// TIA Portal V18 export
// export: Created 2026-01-09T11:31:59.6911216Z, ExportSetting WithDefaults, DisplayName Totally Integrated Automation Portal, DisplayVersion V18 Update 5, DisplayName TIA Portal Openness, DisplayVersion V18 Update 5, DisplayName TIA Portal Teamcenter Gateway, DisplayVersion V18, DisplayName TIA Portal Version Control Interface, DisplayVersion V18, DisplayName SINAMICS Startdrive Advanced, DisplayVersion V18 SP2 Update 1, DisplayName SINAMICS Startdrive G110M, G120, G120C, G120D, G120P, G115D, DisplayVersion V18 SP2 Update 1, DisplayName SINAMICS Startdrive G130, G150, S120, S150, SINAMICS MV, S210, G220, S200, DisplayVersion V18 SP2 Update 1, DisplayName STEP 7 Professional, DisplayVersion V18 Update 5, DisplayName STEP 7 Safety, DisplayVersion V18, DisplayName WinCC Professional, DisplayVersion V18 Update 5
TagTable "2Command Mes To PLC_DB501"
  MEStoPLC_Load_Station1PartOK : Bool  (PLC tag MEStoPLC."MES.Load_Station1PartOK", CPU S71500-2PN_TP700, 1 s)
  MEStoPLC_Load_Station1PartNG : Bool  (PLC tag MEStoPLC."MES.Load_Station1PartNG", CPU S71500-2PN_TP700, 1 s)
  MEStoPLC_Load_Station1ReqMesDone : Bool  (PLC tag MEStoPLC."MES.Load_Station1ReqMesDone", CPU S71500-2PN_TP700, 1 s)
  MEStoPLC_Load_Station1Spare : Bool  (PLC tag MEStoPLC.Spare_1, CPU S71500-2PN_TP700, 1 s)
  MEStoPLC_Load_Station1Spare1 : Bool  (PLC tag MEStoPLC."MES.Load_Station2PartOK", CPU S71500-2PN_TP700, 1 s)
  MEStoPLC_Load_Station1Spare2 : Bool  (PLC tag MEStoPLC."MES.Load_Station2PartNG", CPU S71500-2PN_TP700, 1 s)
  MEStoPLC_Load_Station1Spare3 : Bool  (PLC tag MEStoPLC."MES.Load_Station2ReqMesDone", CPU S71500-2PN_TP700, 1 s)
  MEStoPLC_Load_Station1Spare4 : Bool  (PLC tag MEStoPLC.Spare_2, CPU S71500-2PN_TP700, 1 s)
  MEStoPLC_Load_Station2PartOK : Bool  (PLC tag MEStoPLC."MES.Load_Station3PartOK", CPU S71500-2PN_TP700, 1 s)
  MEStoPLC_Load_Station2PartNG : Bool  (PLC tag MEStoPLC."MES.Load_Station3PartNG", CPU S71500-2PN_TP700, 1 s)
  MEStoPLC_Load_Station2ReqMesDone : Bool  (PLC tag MEStoPLC."MES.Load_Station3ReqMesDone", CPU S71500-2PN_TP700, 1 s)
  MEStoPLC_Load_Station2Spare : Bool  (PLC tag MEStoPLC.Spare_3, CPU S71500-2PN_TP700, 1 s)
  MEStoPLC_Load_Station2Spare1 : Bool  (PLC tag MEStoPLC."MES.Load_Station4PartOK", CPU S71500-2PN_TP700, 1 s)
  MEStoPLC_Load_Station2Spare2 : Bool  (PLC tag MEStoPLC."MES.Load_Station4PartNG", CPU S71500-2PN_TP700, 1 s)
  MEStoPLC_Load_Station2Spare3 : Bool  (PLC tag MEStoPLC."MES.Load_Station4ReqMesDone", CPU S71500-2PN_TP700, 1 s)
  MEStoPLC_Load_Station2Spare4 : Bool  (PLC tag MEStoPLC.Spare_4, CPU S71500-2PN_TP700, 1 s)
  MEStoPLC_Load_Station3PartOK : Bool  (PLC tag MEStoPLC."MES.Load_Station5PartOK", CPU S71500-2PN_TP700, 1 s)
  MEStoPLC_Load_Station3PartNG : Bool  (PLC tag MEStoPLC."MES.Load_Station5PartNG", CPU S71500-2PN_TP700, 1 s)
  MEStoPLC_Load_Station3ReqMesDone : Bool  (PLC tag MEStoPLC."MES.Load_Station5ReqMesDone", CPU S71500-2PN_TP700, 1 s)
  MEStoPLC_Load_Station3Spare : Bool  (PLC tag MEStoPLC.Spare_5, CPU S71500-2PN_TP700, 1 s)
  MEStoPLC_Load_Station3Spare1 : Bool  (PLC tag MEStoPLC."MES.Load_Station6PartOK", CPU S71500-2PN_TP700, 1 s)
  MEStoPLC_Load_Station3Spare2 : Bool  (PLC tag MEStoPLC."MES.Load_Station6PartNG", CPU S71500-2PN_TP700, 1 s)
  MEStoPLC_Load_Station3Spare3 : Bool  (PLC tag MEStoPLC."MES.Load_Station6ReqMesDone", CPU S71500-2PN_TP700, 1 s)
  MEStoPLC_Load_Station3Spare4 : Bool  (PLC tag MEStoPLC.Spare_6, CPU S71500-2PN_TP700, 1 s)
  MEStoPLC_Load_Station4PartOK : Bool  (PLC tag MEStoPLC."MES.Load_Station7PartOK", CPU S71500-2PN_TP700, 1 s)
  MEStoPLC_Load_Station4PartNG : Bool  (PLC tag MEStoPLC."MES.Load_Station7PartNG", CPU S71500-2PN_TP700, 1 s)
  MEStoPLC_Load_Station4ReqMesDone : Bool  (PLC tag MEStoPLC."MES.Load_Station7ReqMesDone", CPU S71500-2PN_TP700, 1 s)
  MEStoPLC_Load_Station4Spare : Bool  (PLC tag MEStoPLC.Spare_7, CPU S71500-2PN_TP700, 1 s)
  MEStoPLC_Load_Station4Spare1 : Bool  (PLC tag MEStoPLC."MES.Load_Station8PartOK", CPU S71500-2PN_TP700, 1 s)
  MEStoPLC_Load_Station4Spare2 : Bool  (PLC tag MEStoPLC."MES.Load_Station8PartNG", CPU S71500-2PN_TP700, 1 s)
  MEStoPLC_Load_Station4Spare3 : Bool  (PLC tag MEStoPLC."MES.Load_Station8ReqMesDone", CPU S71500-2PN_TP700, 1 s)
  MEStoPLC_Load_Station4Spare4 : Bool  (PLC tag MEStoPLC.Spare_8, CPU S71500-2PN_TP700, 1 s)
  MEStoPLC_Load_Station5PartOK : Bool  (PLC tag MEStoPLC.Spare_9, CPU S71500-2PN_TP700, 1 s)
  MEStoPLC_Load_Station5PartNG : Bool  (PLC tag MEStoPLC.Static_3, CPU S71500-2PN_TP700, 1 s)
  MEStoPLC_Load_Station5ReqMesDone : Bool  (PLC tag MEStoPLC."MES.Load_SubPart1OK", CPU S71500-2PN_TP700, 1 s)
  MEStoPLC_Load_Station5Spare : Bool  (PLC tag MEStoPLC."MES.Load_SubPart1tNG", CPU S71500-2PN_TP700, 1 s)
  MEStoPLC_Load_Station5Spare1 : Bool  (PLC tag MEStoPLC."MES.Load_SubPart1ReqMesDone", CPU S71500-2PN_TP700, 1 s)
  MEStoPLC_Load_Station5Spare2 : Bool  (PLC tag MEStoPLC.Spare_10, CPU S71500-2PN_TP700, 1 s)
  MEStoPLC_Load_Station5Spare3 : Bool  (PLC tag MEStoPLC."MES.Load_SubPart2OK", CPU S71500-2PN_TP700, 1 s)
  MEStoPLC_Load_Station5Spare4 : Bool  (PLC tag MEStoPLC."MES.Load_SubPart2tNG", CPU S71500-2PN_TP700, 1 s)
  MEStoPLC_Load_Station6PartOK : Bool  (PLC tag MEStoPLC."MES.Load_SubPart2ReqMesDone", CPU S71500-2PN_TP700, 1 s)
  MEStoPLC_Load_Station6PartNG : Bool  (PLC tag MEStoPLC.Spare_11, CPU S71500-2PN_TP700, 1 s)
  MEStoPLC_Load_Station6ReqMesDone : Bool  (PLC tag MEStoPLC."MES.Load_SubPart3OK", CPU S71500-2PN_TP700, 1 s)
  MEStoPLC_Load_Station6Spare : Bool  (PLC tag MEStoPLC."MES.Load_SubPart3tNG", CPU S71500-2PN_TP700, 1 s)
  MEStoPLC_Load_Station6Spare1 : Bool  (PLC tag MEStoPLC."MES.Load_SubPart3ReqMesDone", CPU S71500-2PN_TP700, 1 s)
  MEStoPLC_Load_Station6Spare2 : Bool  (PLC tag MEStoPLC.Spare_12, CPU S71500-2PN_TP700, 1 s)
  MEStoPLC_Load_Station6Spare3 : Bool  (PLC tag MEStoPLC."MES.Load_SubPart4OK", CPU S71500-2PN_TP700, 1 s)
  MEStoPLC_Load_Station6Spare4 : Bool  (PLC tag MEStoPLC."MES.Load_SubPart4tNG", CPU S71500-2PN_TP700, 1 s)
  MEStoPLC_Load_Station7PartOK : Bool  (PLC tag MEStoPLC."MES.Load_SubPart4ReqMesDone", CPU S71500-2PN_TP700, 1 s)
  MEStoPLC_Load_Station7PartNG : Bool  (PLC tag MEStoPLC.Spare_13, CPU S71500-2PN_TP700, 1 s)
  MEStoPLC_Load_Station7ReqMesDone : Bool  (PLC tag MEStoPLC."MES.Load_SubPart5OK", CPU S71500-2PN_TP700, 1 s)
  MEStoPLC_Load_Station7Spare : Bool  (PLC tag MEStoPLC."MES.Load_SubPart5tNG", CPU S71500-2PN_TP700, 1 s)
  MEStoPLC_Load_Station7Spare1 : Bool  (PLC tag MEStoPLC."MES.Load_SubPart5ReqMesDone", CPU S71500-2PN_TP700, 1 s)
  MEStoPLC_Load_Station7Spare2 : Bool  (PLC tag MEStoPLC.Spare_14, CPU S71500-2PN_TP700, 1 s)
  MEStoPLC_Load_Station7Spare3 : Bool  (PLC tag MEStoPLC."MES.Load_SubPart6OK", CPU S71500-2PN_TP700, 1 s)
  MEStoPLC_Load_Station7Spare4 : Bool  (PLC tag MEStoPLC."MES.Load_SubPart6tNG", CPU S71500-2PN_TP700, 1 s)
  MEStoPLC_Load_Station8PartOK : Bool  (PLC tag MEStoPLC."MES.Load_SubPart6ReqMesDone", CPU S71500-2PN_TP700, 1 s)
  MEStoPLC_Load_Station8PartNG : Bool  (PLC tag MEStoPLC.Spare_15, CPU S71500-2PN_TP700, 1 s)
  MEStoPLC_Load_Station8ReqMesDone : Bool  (PLC tag MEStoPLC."MES.Load_SubPart7OK", CPU S71500-2PN_TP700, 1 s)
  MEStoPLC_Load_Station8Spare : Bool  (PLC tag MEStoPLC."MES.Load_SubPart7tNG", CPU S71500-2PN_TP700, 1 s)
  MEStoPLC_Load_Station8Spare5 : Bool  (PLC tag MEStoPLC."MES.Load_SubPart7ReqMesDone", CPU S71500-2PN_TP700, 1 s)
  MEStoPLC_Load_Station8Spare6 : Bool  (PLC tag MEStoPLC.Spare_16, CPU S71500-2PN_TP700, 1 s)
  MEStoPLC_Load_Station8Spare8 : Bool  (PLC tag MEStoPLC."MES.Load_SubPart8OK", CPU S71500-2PN_TP700, 1 s)
  MEStoPLC_Load_Station8Spare9 : Bool  (PLC tag MEStoPLC."MES.Load_SubPart8tNG", CPU S71500-2PN_TP700, 1 s)
  MEStoPLC_Load_SubPart1OK : Bool  (PLC tag MEStoPLC.Spare, CPU S71500-2PN_TP700, 1 s)
  MEStoPLC_Load_SubPart1tNG : Bool  (PLC tag MEStoPLC.Spare_17, CPU S71500-2PN_TP700, 1 s)
  MEStoPLC_Load_SubPart1ReqMesDone : Bool  (PLC tag MEStoPLC."MES.Load_ResultsStored1OK", CPU S71500-2PN_TP700, 1 s)
  MEStoPLC_Load_SubPart2OK : Bool  (PLC tag MEStoPLC."MES.Load_ResultsStored2ReqMesDone", CPU S71500-2PN_TP700, 1 s)
  MEStoPLC_Load_SubPart2tNG : Bool  (PLC tag MEStoPLC.Spare_19, CPU S71500-2PN_TP700, 1 s)
  MEStoPLC_Load_SubPart2ReqMesDone : Bool  (PLC tag MEStoPLC."MES.Load_ResultsStored3OK", CPU S71500-2PN_TP700, 1 s)
  MEStoPLC_Load_SubPart3OK : Bool  (PLC tag MEStoPLC."MES.Load_ResultsStored4ReqMesDone", CPU S71500-2PN_TP700, 1 s)
  MEStoPLC_Load_SubPart3tNG : Bool  (PLC tag MEStoPLC.Spare_21, CPU S71500-2PN_TP700, 1 s)
  MEStoPLC_Load_SubPart3ReqMesDone : Bool  (PLC tag MEStoPLC."MES.Load_ResultsStored5OK", CPU S71500-2PN_TP700, 1 s)
  MEStoPLC_Load_SubPart4OK : Bool  (PLC tag MEStoPLC."MES.Load_ResultsStored6ReqMesDone", CPU S71500-2PN_TP700, 1 s)
  MEStoPLC_Load_SubPart4tNG : Bool  (PLC tag MEStoPLC.Spare_23, CPU S71500-2PN_TP700, 1 s)
  MEStoPLC_Load_SubPart4ReqMesDone : Bool  (PLC tag MEStoPLC."MES.Load_ResultsStored7OK", CPU S71500-2PN_TP700, 1 s)
  MEStoPLC_Load_SubPart5OK : Bool  (PLC tag MEStoPLC."MES.Load_ResultsStored8ReqMesDone", CPU S71500-2PN_TP700, 1 s)
  MEStoPLC_Load_SubPart5tNG : Bool  (PLC tag MEStoPLC."MES.Load_StoveCheckInOk", CPU S71500-2PN_TP700, 1 s)
  MEStoPLC_Load_SubPart5ReqMesDone : Bool  (PLC tag MEStoPLC.Static_1, CPU S71500-2PN_TP700, 1 s)
  MEStoPLC_Load_SubPart6OK : Bool  (PLC tag MEStoPLC.Spare_31, CPU S71500-2PN_TP700, 1 s)
  MEStoPLC_Load_SubPart6tNG : Bool  (PLC tag MEStoPLC.Spare_32, CPU S71500-2PN_TP700, 1 s)
  MEStoPLC_Load_SubPart6ReqMesDone : Bool  (PLC tag MEStoPLC.Spare_33, CPU S71500-2PN_TP700, 1 s)
  MEStoPLC_Load_SubPart7OK : Bool  (PLC tag MEStoPLC."MES.Unload_ResultsStored2NG", CPU S71500-2PN_TP700, 1 s)
  MEStoPLC_Load_SubPart7tNG : Bool  (PLC tag MEStoPLC."MES.Unload_ResultsStored2ReqMesDone", CPU S71500-2PN_TP700, 1 s)
  MEStoPLC_Load_SubPart7ReqMesDone : Bool  (PLC tag MEStoPLC.Spare_35, CPU S71500-2PN_TP700, 1 s)
  MEStoPLC_Load_SubPart8OK : Bool  (PLC tag MEStoPLC."MES.Unload_ResultsStored4NG", CPU S71500-2PN_TP700, 1 s)
  MEStoPLC_Load_ResultsStored1OK : Bool  (PLC tag MEStoPLC."MES.Unload_ResultsStored6ReqMesDone", CPU S71500-2PN_TP700, 1 s)
  MEStoPLC_Load_ResultsStored1NG : Bool  (PLC tag MEStoPLC.Spare_39, CPU S71500-2PN_TP700, 1 s)
  MEStoPLC_Load_ResultsStored1ReqMesDone : Bool  (PLC tag MEStoPLC."MES.Unload_ResultsStored7OK", CPU S71500-2PN_TP700, 1 s)
  MEStoPLC_Load_ResultsStored1Spare : Bool  (PLC tag MEStoPLC."MES.Unload_ResultsStored7NG", CPU S71500-2PN_TP700, 1 s)
  MEStoPLC_Load_ResultsStored1Spare1 : Bool  (PLC tag MEStoPLC."MES.Unload_ResultsStored7ReqMesDone", CPU S71500-2PN_TP700, 1 s)
  MEStoPLC_Load_ResultsStored1Spare2 : Bool  (PLC tag MEStoPLC.Spare_40, CPU S71500-2PN_TP700, 1 s)
  MEStoPLC_Load_ResultsStored1Spare3 : Bool  (PLC tag MEStoPLC."MES.Unload_ResultsStored8OK", CPU S71500-2PN_TP700, 1 s)
  MEStoPLC_Load_ResultsStored1Spare4 : Bool  (PLC tag MEStoPLC."MES.Unload_ResultsStored8NG", CPU S71500-2PN_TP700, 1 s)
  MEStoPLC_Load_ResultsStored2OK : Bool  (PLC tag MEStoPLC."MES.Unload_ResultsStored8ReqMesDone", CPU S71500-2PN_TP700, 1 s)
  MEStoPLC_Load_ResultsStored2NG : Bool  (PLC tag MEStoPLC.Spare_41, CPU S71500-2PN_TP700, 1 s)
  MEStoPLC_Load_ResultsStored2ReqMesDone : Bool  (PLC tag MEStoPLC."MES.HeartbeatSignal", CPU S71500-2PN_TP700, 1 s)
